FUNCTION Scale : LREAL
VAR_INPUT
	signal : LREAL;
	inputMin : LREAL;
	inputMax : LREAL;
	outputMin : LREAL;
	outputMax : LREAL;
END_VAR
VAR
END_VAR

IF signal < inputMin OR signal > inputMax THEN
	Scale := 0;
ELSE
	IF ((inputMax - inputMin) + outputMin) <> 0 THEN
	    Scale := ((signal - inputMin) * (outputMax - outputMin) / (inputMax - inputMin) + outputMin);
	ELSE
		Scale := 0;
	END_IF
END_IF

END_FUNCTION

(* stored: Version 1.1.0.1, ProductVersion 3.1.4024.9
   POU Scale: Id {4b96f4d6-2f77-4c1d-94c4-2f359e2a6940}, SpecialFunc None *)
